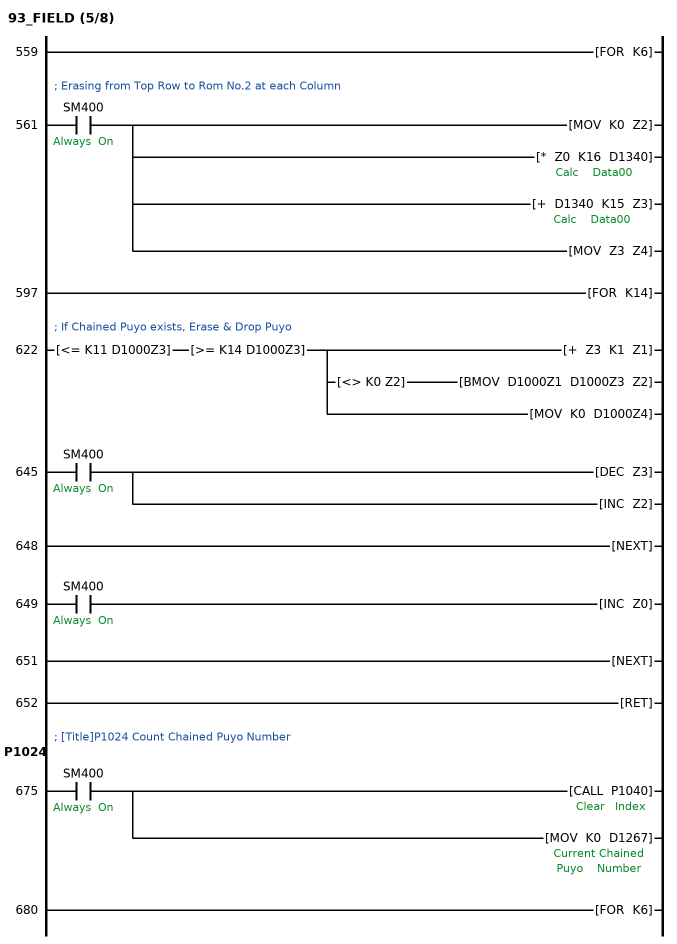
[picture p24: ladder of 93_FIELD, rungs at steps 559 to 680]
; Start Erasing at Column No.2 ,and End at No.7
559   FOR     K6
561   LD      SM400  ; Always  On
      MOV     K0 Z2
      *       Z0 K16 D1340
      +       D1340 K15 Z3
      MOV     Z3 Z4
; Erasing from Top Row to Rom No.2 at each Column
597   FOR     K14
; If Chained Puyo exists, Erase & Drop Puyo
622   LD<=    K11 D1000Z3
      AND>=   K14 D1000Z3
      +       Z3 K1 Z1
      MPS
      AND<>   K0 Z2
      BMOV    D1000Z1 D1000Z3 Z2
      MPP
      MOV     K0 D1000Z4
645   LD      SM400  ; Always  On
      DEC     Z3
      INC     Z2
648   NEXT
649   LD      SM400  ; Always  On
      INC     Z0
651   NEXT
652   RET
; [Title]P1024 Count Chained Puyo Number
      P1024
675   LD      SM400  ; Always  On
      CALL    P1040
      MOV     K0 D1267  ; Current Chained Puyo    Number
680   FOR     K6
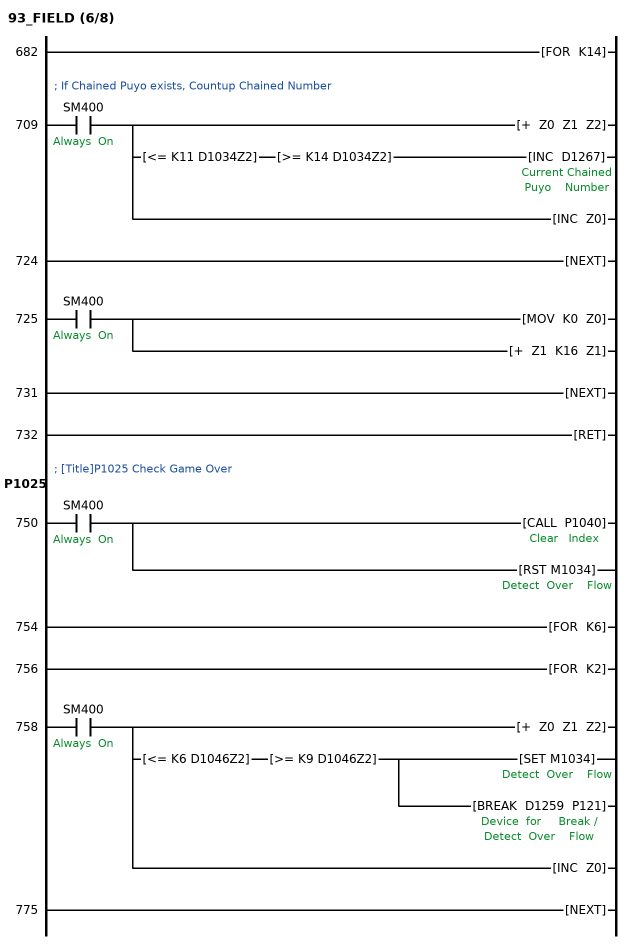
682   FOR     K14
; If Chained Puyo exists, Countup Chained Number
709   LD      SM400  ; Always  On
      +       Z0 Z1 Z2
      MPS
      AND<=   K11 D1034Z2
      AND>=   K14 D1034Z2
      INC     D1267
      MPP
      INC     Z0
724   NEXT
725   LD      SM400  ; Always  On
      MOV     K0 Z0
      +       Z1 K16 Z1
731   NEXT
732   RET
; [Title]P1025 Check Game Over
      P1025
750   LD      SM400  ; Always  On
      CALL    P1040
      RST     M1034  ; Detect  Over    Flow
754   FOR     K6
756   FOR     K2
758   LD      SM400  ; Always  On
      +       Z0 Z1 Z2
      MPS
      AND<=   K6 D1046Z2
      AND>=   K9 D1046Z2
      SET     M1034  ; Detect  Over    Flow
      BREAK   D1259 P121  ; Device  for     Break / Detect  Over    Flow
      MPP
      INC     Z0
775   NEXT
      P121
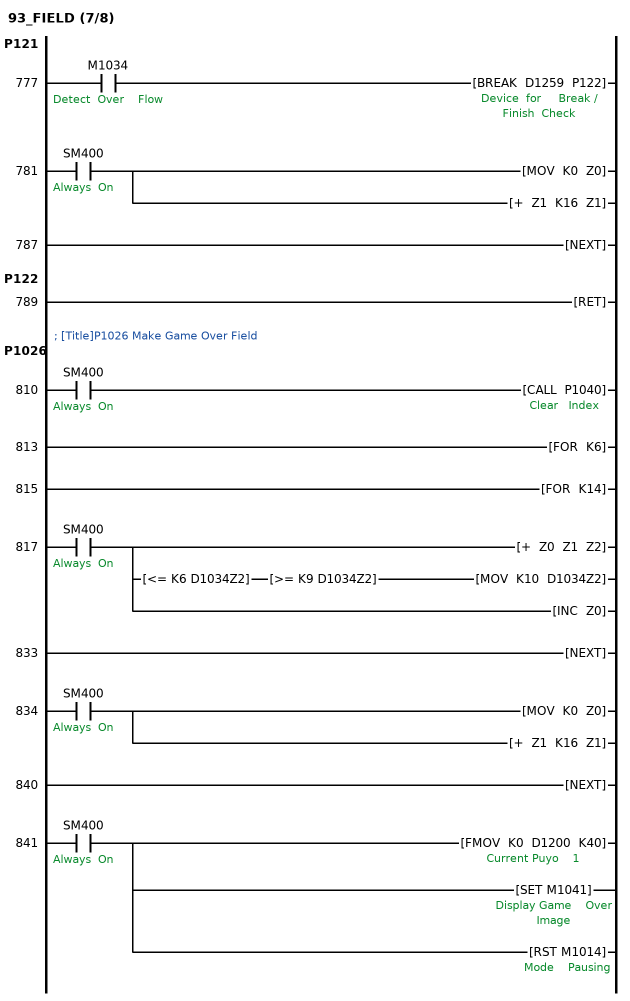
777   LD      M1034  ; Detect  Over    Flow
      BREAK   D1259 P122  ; Finish  Check
781   LD      SM400  ; Always  On
      MOV     K0 Z0
      +       Z1 K16 Z1
787   NEXT
      P122
789   RET
; [Title]P1026 Make Game Over Field
      P1026
810   LD      SM400  ; Always  On
      CALL    P1040
813   FOR     K6
815   FOR     K14
817   LD      SM400  ; Always  On
      +       Z0 Z1 Z2
      MPS
      AND<=   K6 D1034Z2
      AND>=   K9 D1034Z2
      MOV     K10 D1034Z2
      MPP
      INC     Z0
833   NEXT
834   LD      SM400  ; Always  On
      MOV     K0 Z0
      +       Z1 K16 Z1
840   NEXT
841   LD      SM400  ; Always  On
      FMOV    K0 D1200 K40  ; Current Puyo    1
      SET     M1041  ; Display Game    Over    Image
      RST     M1014  ; Mode    Pausing
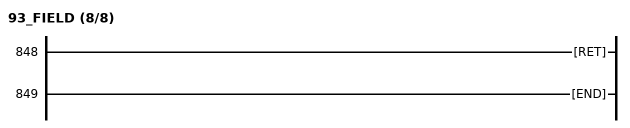
848   RET
849   END
END_PROGRAM

PROGRAM 94_MOVE  // Move Puyo Operation
; [Title]P1030 Move to Left Puyo
      P1030
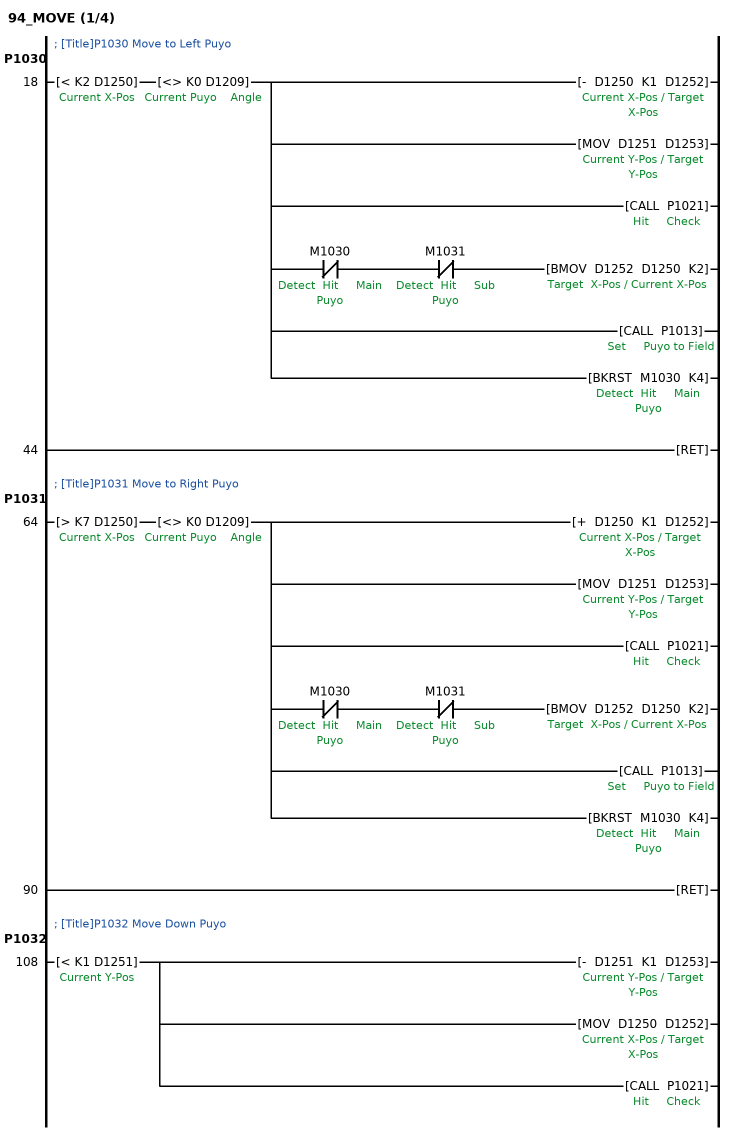
18    LD<     K2 D1250  ; Current X-Pos
      AND<>   K0 D1209  ; Current Puyo    Angle
      -       D1250 K1 D1252  ; Target  X-Pos
      MOV     D1251 D1253  ; Current Y-Pos / Target  Y-Pos
      CALL    P1021  ; Hit     Check
      MPS
      ANI     M1030  ; Detect  Hit     Main    Puyo
      ANI     M1031  ; Detect  Hit     Sub     Puyo
      BMOV    D1252 D1250 K2
      MPP
      CALL    P1013  ; Set     Puyo to Field
      BKRST   M1030 K4
44    RET
; [Title]P1031 Move to Right Puyo
      P1031
64    LD>     K7 D1250  ; Current X-Pos
      AND<>   K0 D1209  ; Current Puyo    Angle
      +       D1250 K1 D1252
      MOV     D1251 D1253
      CALL    P1021
      MPS
      ANI     M1030  ; Detect  Hit     Main    Puyo
      ANI     M1031  ; Detect  Hit     Sub     Puyo
      BMOV    D1252 D1250 K2
      MPP
      CALL    P1013
      BKRST   M1030 K4
90    RET
; [Title]P1032 Move Down Puyo
      P1032
108   LD<     K1 D1251  ; Current Y-Pos
      -       D1251 K1 D1253
      MOV     D1250 D1252
      CALL    P1021
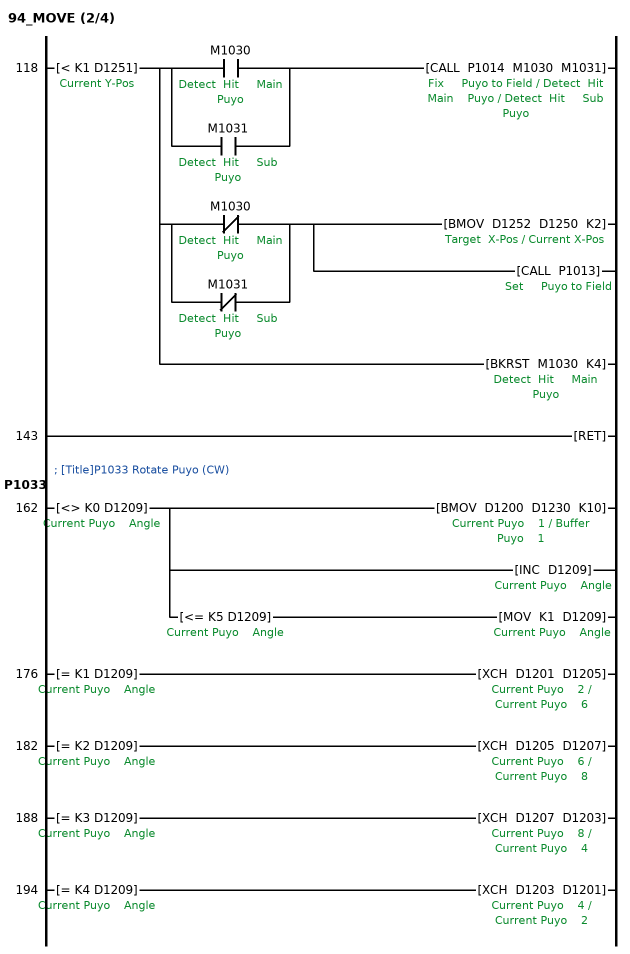
118   LD<     K1 D1251  ; Current Y-Pos
      MPS
      LD      M1030  ; Detect  Hit     Main    Puyo
      OR      M1031  ; Detect  Hit     Sub     Puyo
      ANB
      CALL    P1014 M1030 M1031  ; Fix     Puyo to Field
      MRD
      LDI     M1030  ; Detect  Hit     Main    Puyo
      ORI     M1031  ; Detect  Hit     Sub     Puyo
      ANB
      BMOV    D1252 D1250 K2
      CALL    P1013
      MPP
      BKRST   M1030 K4
143   RET
; [Title]P1033 Rotate Puyo (CW)
      P1033
162   LD<>    K0 D1209  ; Current Puyo    Angle
      BMOV    D1200 D1230 K10  ; Current Puyo    1 / Buffer  Puyo    1
      INC     D1209
      AND<=   K5 D1209  ; Current Puyo    Angle
      MOV     K1 D1209
176   LD=     K1 D1209  ; Current Puyo    Angle
      XCH     D1201 D1205  ; Current Puyo    2 / Current Puyo    6
182   LD=     K2 D1209  ; Current Puyo    Angle
      XCH     D1205 D1207  ; Current Puyo    8
188   LD=     K3 D1209  ; Current Puyo    Angle
      XCH     D1207 D1203  ; Current Puyo    4
194   LD=     K4 D1209  ; Current Puyo    Angle
      XCH     D1203 D1201
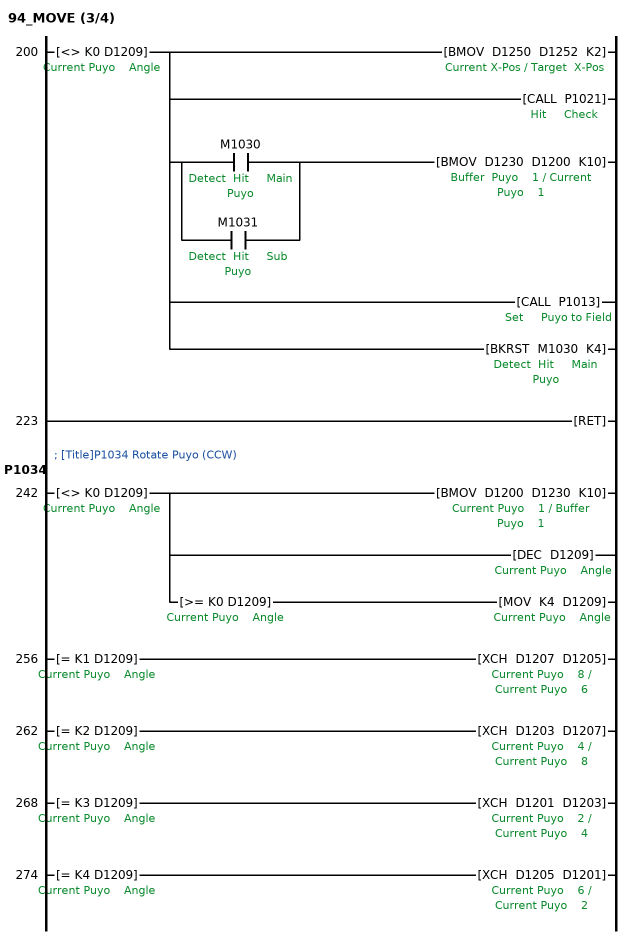
200   LD<>    K0 D1209  ; Current Puyo    Angle
      BMOV    D1250 D1252 K2
      CALL    P1021
      MPS
      LD      M1030  ; Detect  Hit     Main    Puyo
      OR      M1031  ; Detect  Hit     Sub     Puyo
      ANB
      BMOV    D1230 D1200 K10
      MPP
      CALL    P1013
      BKRST   M1030 K4
223   RET
; [Title]P1034 Rotate Puyo (CCW)
      P1034
242   LD<>    K0 D1209  ; Current Puyo    Angle
      BMOV    D1200 D1230 K10
      DEC     D1209
      AND>=   K0 D1209  ; Current Puyo    Angle
      MOV     K4 D1209
256   LD=     K1 D1209  ; Current Puyo    Angle
      XCH     D1207 D1205
262   LD=     K2 D1209  ; Current Puyo    Angle
      XCH     D1203 D1207
268   LD=     K3 D1209  ; Current Puyo    Angle
      XCH     D1201 D1203
274   LD=     K4 D1209  ; Current Puyo    Angle
      XCH     D1205 D1201
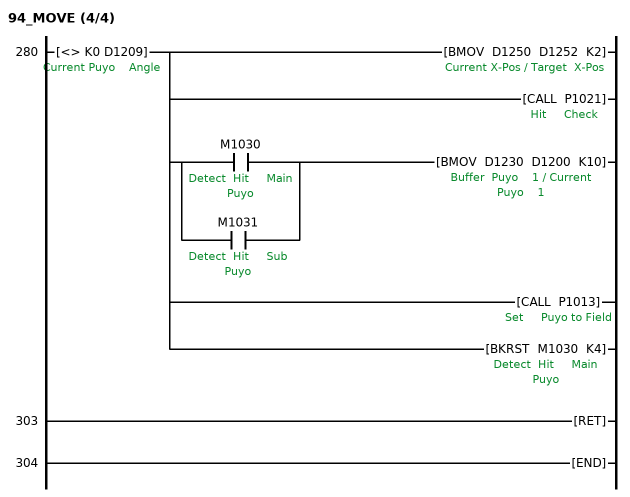
280   LD<>    K0 D1209  ; Current Puyo    Angle
      BMOV    D1250 D1252 K2
      CALL    P1021
      MPS
      LD      M1030  ; Detect  Hit     Main    Puyo
      OR      M1031  ; Detect  Hit     Sub     Puyo
      ANB
      BMOV    D1230 D1200 K10
      MPP
      CALL    P1013
      BKRST   M1030 K4
303   RET
304   END
END_PROGRAM

PROGRAM 02_GAME  // Game Main
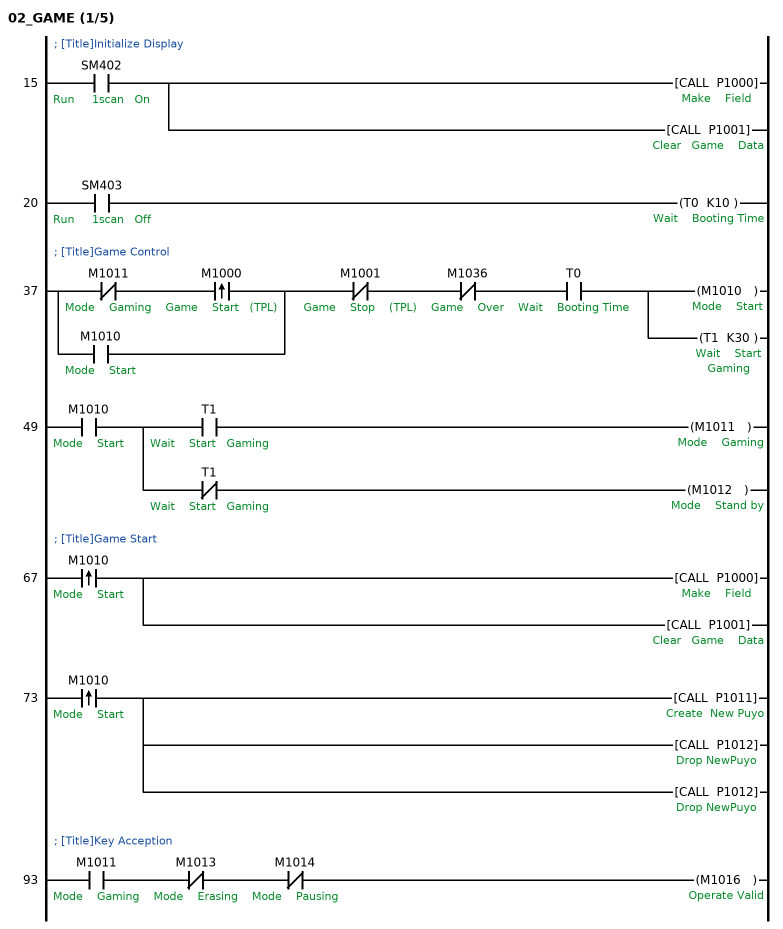
; [Title]Initialize Display
15    LD      SM402  ; Run     1scan   On
      CALL    P1000  ; Make    Field
      CALL    P1001  ; Clear   Game    Data
20    LD      SM403  ; Run     1scan   Off
      OUT     T0 K10  ; Wait    Booting Time
; [Title]Game Control
37    LDI     M1011  ; Mode    Gaming
      ANDP    M1000  ; Game    Start   (TPL)
      OR      M1010  ; Mode    Start
      ANI     M1001  ; Game    Stop    (TPL)
      ANI     M1036  ; Game    Over
      AND     T0  ; Wait    Booting Time
      OUT     M1010  ; Mode    Start
      OUT     T1 K30  ; Wait    Start   Gaming
49    LD      M1010  ; Mode    Start
      MPS
      AND     T1  ; Wait    Start   Gaming
      OUT     M1011  ; Mode    Gaming
      MPP
      ANI     T1  ; Wait    Start   Gaming
      OUT     M1012  ; Mode    Stand by
; [Title]Game Start
67    LDP     M1010  ; Mode    Start
      CALL    P1000
      CALL    P1001
73    LDP     M1010  ; Mode    Start
      CALL    P1011  ; Create  New Puyo
      CALL    P1012  ; Drop NewPuyo
      CALL    P1012
; [Title]Key Acception
93    LD      M1011  ; Mode    Gaming
      ANI     M1013  ; Mode    Erasing
      ANI     M1014  ; Mode    Pausing
      OUT     M1016  ; Operate Valid
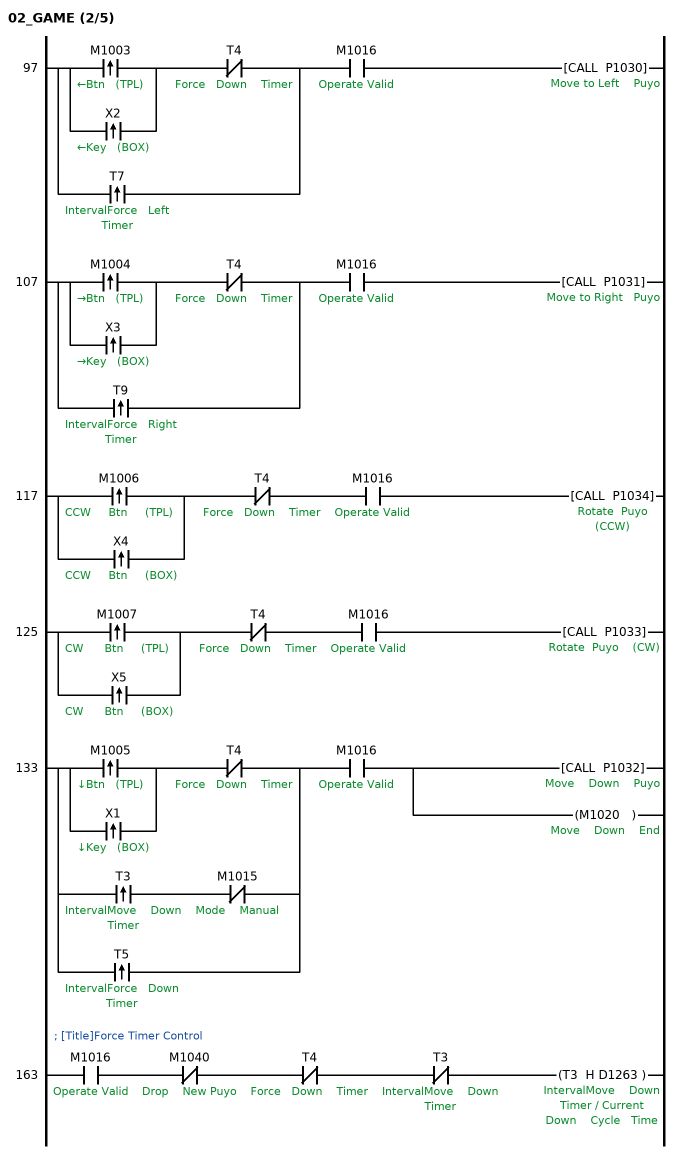
97    LDP     M1003  ; ←Btn   (TPL)
      ORP     X2  ; ←Key   (BOX)
      ANI     T4  ; Force   Down    Timer
      ORP     T7  ; IntervalForce   Left    Timer
      AND     M1016  ; Operate Valid
      CALL    P1030  ; Move to Left    Puyo
107   LDP     M1004  ; →Btn   (TPL)
      ORP     X3  ; →Key   (BOX)
      ANI     T4  ; Force   Down    Timer
      ORP     T9  ; IntervalForce   Right   Timer
      AND     M1016  ; Operate Valid
      CALL    P1031  ; Move to Right   Puyo
117   LDP     M1006  ; CCW     Btn     (TPL)
      ORP     X4  ; CCW     Btn     (BOX)
      ANI     T4  ; Force   Down    Timer
      AND     M1016  ; Operate Valid
      CALL    P1034  ; Rotate  Puyo    (CCW)
125   LDP     M1007  ; CW      Btn     (TPL)
      ORP     X5  ; CW      Btn     (BOX)
      ANI     T4  ; Force   Down    Timer
      AND     M1016  ; Operate Valid
      CALL    P1033  ; Rotate  Puyo    (CW)
133   LDP     M1005  ; ↓Btn   (TPL)
      ORP     X1  ; ↓Key   (BOX)
      ANI     T4  ; Force   Down    Timer
      LDP     T3  ; IntervalMove    Down    Timer
      ANI     M1015  ; Mode    Manual
      ORB
      ORP     T5  ; IntervalForce   Down    Timer
      AND     M1016  ; Operate Valid
      CALL    P1032  ; Move    Down    Puyo
      OUT     M1020  ; Move    Down    End
; [Title]Force Timer Control
163   LD      M1016  ; Operate Valid
      ANI     M1040  ; Drop    New Puyo
      ANI     T4  ; Force   Down    Timer
      ANI     T3  ; IntervalMove    Down    Timer
      OUTH    T3 D1263  ; IntervalMove    Down    Timer / Current Down    Cycle   Time
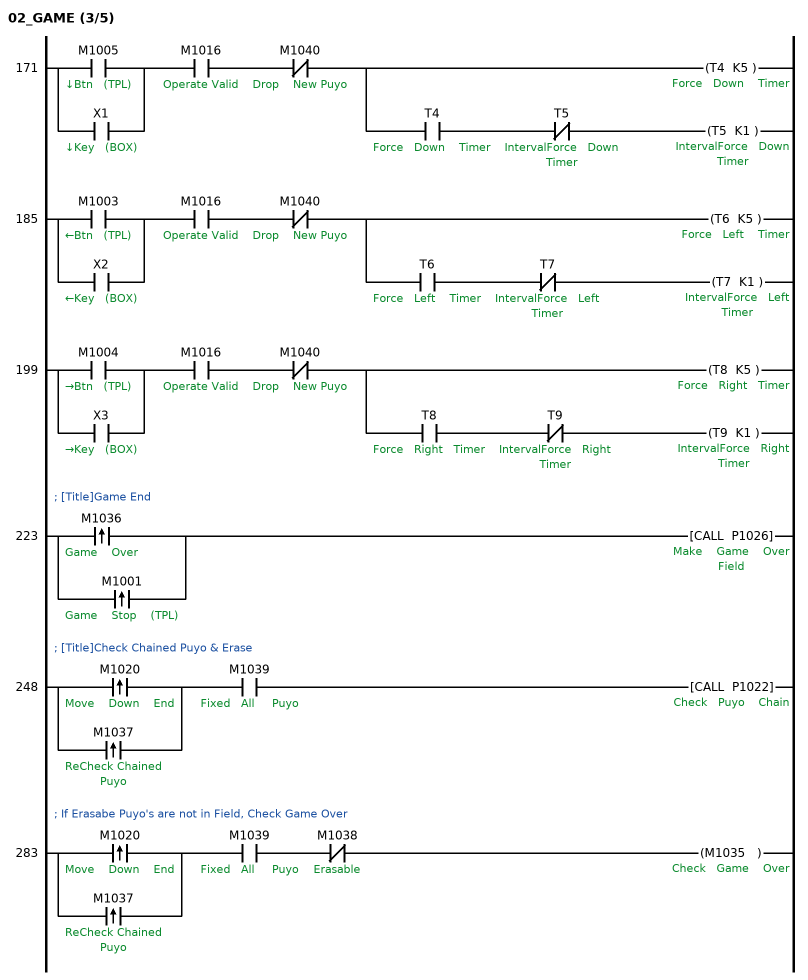
171   LD      M1005  ; ↓Btn   (TPL)
      OR      X1  ; ↓Key   (BOX)
      AND     M1016  ; Operate Valid
      ANI     M1040  ; Drop    New Puyo
      OUT     T4 K5  ; Force   Down    Timer
      AND     T4  ; Force   Down    Timer
      ANI     T5  ; IntervalForce   Down    Timer
      OUT     T5 K1  ; IntervalForce   Down    Timer
185   LD      M1003  ; ←Btn   (TPL)
      OR      X2  ; ←Key   (BOX)
      AND     M1016  ; Operate Valid
      ANI     M1040  ; Drop    New Puyo
      OUT     T6 K5  ; Force   Left    Timer
      AND     T6  ; Force   Left    Timer
      ANI     T7  ; IntervalForce   Left    Timer
      OUT     T7 K1  ; IntervalForce   Left    Timer
199   LD      M1004  ; →Btn   (TPL)
      OR      X3  ; →Key   (BOX)
      AND     M1016  ; Operate Valid
      ANI     M1040  ; Drop    New Puyo
      OUT     T8 K5  ; Force   Right   Timer
      AND     T8  ; Force   Right   Timer
      ANI     T9  ; IntervalForce   Right   Timer
      OUT     T9 K1  ; IntervalForce   Right   Timer
; [Title]Game End
223   LDP     M1036  ; Game    Over
      ORP     M1001  ; Game    Stop    (TPL)
      CALL    P1026  ; Make    Game    Over    Field
; [Title]Check Chained Puyo & Erase
248   LDP     M1020  ; Move    Down    End
      ORP     M1037  ; ReCheck Chained Puyo
      AND     M1039  ; Fixed   All     Puyo
      CALL    P1022  ; Check   Puyo    Chain
; If Erasabe Puyo's are not in Field, Check Game Over
283   LDP     M1020  ; Move    Down    End
      ORP     M1037  ; ReCheck Chained Puyo
      AND     M1039  ; Fixed   All     Puyo
      ANI     M1038  ; Erasable
      OUT     M1035  ; Check   Game    Over
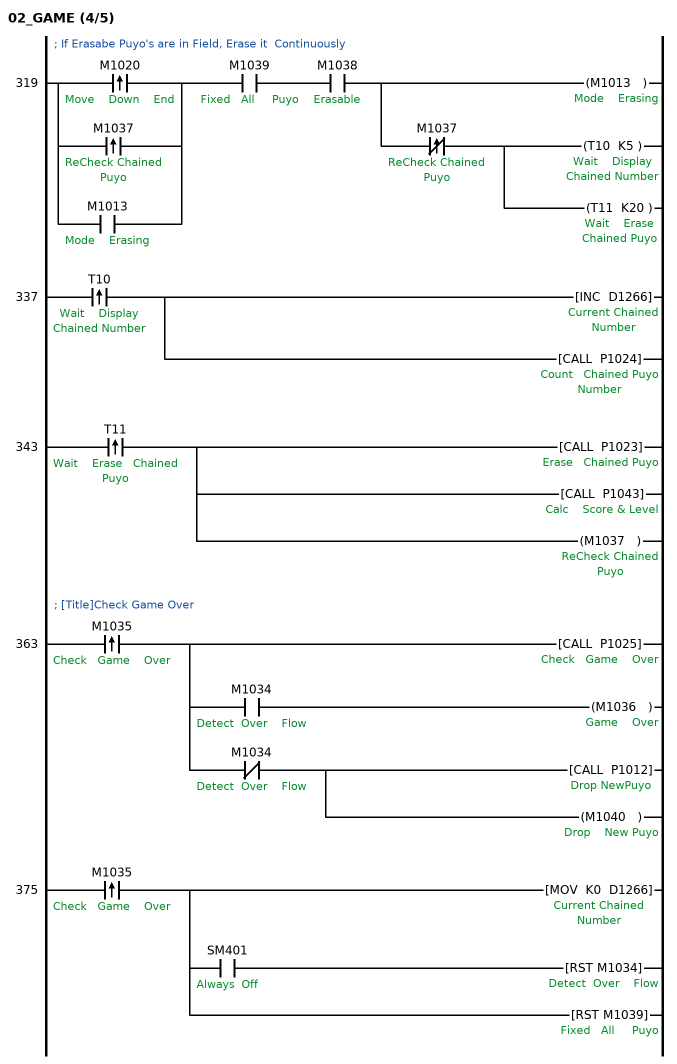
; If Erasabe Puyo's are in Field, Erase it  Continuously
319   LDP     M1020  ; Move    Down    End
      ORP     M1037  ; ReCheck Chained Puyo
      OR      M1013  ; Mode    Erasing
      AND     M1039  ; Fixed   All     Puyo
      AND     M1038  ; Erasable
      OUT     M1013  ; Mode    Erasing
      ANDPI   M1037  ; ReCheck Chained Puyo
      OUT     T10 K5  ; Wait    Display Chained Number
      OUT     T11 K20  ; Wait    Erase   Chained Puyo
337   LDP     T10  ; Wait    Display Chained Number
      INC     D1266  ; Current Chained Number
      CALL    P1024  ; Count   Chained Puyo    Number
343   LDP     T11  ; Wait    Erase   Chained Puyo
      CALL    P1023  ; Erase   Chained Puyo
      CALL    P1043  ; Calc    Score & Level
      OUT     M1037  ; ReCheck Chained Puyo
; [Title]Check Game Over
363   LDP     M1035  ; Check   Game    Over
      CALL    P1025  ; Check   Game    Over
      MPS
      AND     M1034  ; Detect  Over    Flow
      OUT     M1036  ; Game    Over
      MPP
      ANI     M1034  ; Detect  Over    Flow
      CALL    P1012
      OUT     M1040  ; Drop    New Puyo
375   LDP     M1035  ; Check   Game    Over
      MOV     K0 D1266
      MPS
      AND     SM401  ; Always  Off
      RST     M1034  ; Detect  Over    Flow
      MPP
      RST     M1039  ; Fixed   All     Puyo
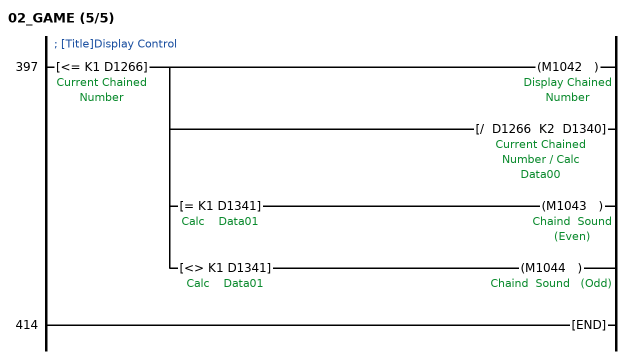
; [Title]Display Control
397   LD<=    K1 D1266  ; Current Chained Number
      OUT     M1042  ; Display Chained Number
      /       D1266 K2 D1340  ; Calc    Data00
      MPS
      AND=    K1 D1341  ; Calc    Data01
      OUT     M1043  ; Chaind  Sound   (Even)
      MPP
      AND<>   K1 D1341  ; Calc    Data01
      OUT     M1044  ; Chaind  Sound   (Odd)
414   END
END_PROGRAM

// device comments not shown above
D1034  ; Field   02, 02
M1017  ; Disable Free    Fall    Puyo
M1053  ; ==DBG== Trigger Setup   04
M1054  ; ==DBG== Trigger Setup   05
M1055  ; ==DBG== Trigger Setup   06
M1056  ; ==DBG== Trigger Setup   07
M1057  ; ==DBG== Trigger Setup   08
M1058  ; ==DBG== Trigger Setup   09
M1059  ; ==DBG== Trigger Setup   10
M1065  ; ==DBG== Trigger Puyo    06
M1066  ; ==DBG== Trigger Puyo    07
M1067  ; ==DBG== Trigger Puyo    08
M1068  ; ==DBG== Trigger Puyo    09
M1069  ; ==DBG== Trigger Puyo    10
M1077  ; ==DBG== Trigger Field   08
M1078  ; ==DBG== Trigger Field   09
M1079  ; ==DBG== Trigger Field   10
M1085  ; ==DBG== Trigger Move    06
M1086  ; ==DBG== Trigger Move    07
M1087  ; ==DBG== Trigger Move    08
M1088  ; ==DBG== Trigger Move    09
M1089  ; ==DBG== Trigger Move    10
M1095  ; ==DBG== Trigger Tools   06
M1096  ; ==DBG== Trigger Tools   07
M1097  ; ==DBG== Trigger Tools   08
M1098  ; ==DBG== Trigger Tools   09
M1099  ; ==DBG== Trigger Tools   10
P11  ; Create  New Puyo
D1001  ; Field   00, 01
D1002  ; Field   00, 02
D1003  ; Field   00, 03
D1004  ; Field   00, 04
D1005  ; Field   00, 05
D1006  ; Field   00, 06
D1007  ; Field   00, 07
D1008  ; Field   00, 08
D1009  ; Field   00, 09
D1010  ; Field   00, 10
D1011  ; Field   00, 11
D1012  ; Field   00, 12
D1013  ; Field   00, 13
D1014  ; Field   00, 14
D1015  ; Field   00, 15
D1016  ; Field   01, 00
D1017  ; Field   01, 01
D1018  ; Field   01, 02
D1019  ; Field   01, 03
D1020  ; Field   01, 04
D1021  ; Field   01, 05
D1022  ; Field   01, 06
D1023  ; Field   01, 07
D1024  ; Field   01, 08
D1025  ; Field   01, 09
D1026  ; Field   01, 10
D1027  ; Field   01, 11
D1028  ; Field   01, 12
D1029  ; Field   01, 13
D1030  ; Field   01, 14
D1031  ; Field   01, 15
D1033  ; Field   02, 01
D1035  ; Field   02, 03
D1036  ; Field   02, 04
D1037  ; Field   02, 05
D1038  ; Field   02, 06
D1039  ; Field   02, 07
D1040  ; Field   02, 08
D1041  ; Field   02, 09
D1042  ; Field   02, 10
D1043  ; Field   02, 11
D1044  ; Field   02, 12
D1045  ; Field   02, 13
D1046  ; Field   02, 14
D1047  ; Field   02, 15
D1048  ; Field   03, 00
D1049  ; Field   03, 01
D1050  ; Field   03, 02
D1051  ; Field   03, 03
D1052  ; Field   03, 04
D1053  ; Field   03, 05
D1054  ; Field   03, 06
D1055  ; Field   03, 07
D1056  ; Field   03, 08
D1057  ; Field   03, 09
D1058  ; Field   03, 10
D1059  ; Field   03, 11
D1060  ; Field   03, 12
D1061  ; Field   03, 13
D1062  ; Field   03, 14
D1063  ; Field   03, 15
D1064  ; Field   04, 00
D1065  ; Field   04, 01
D1066  ; Field   04, 02
D1067  ; Field   04, 03
D1068  ; Field   04, 04
D1069  ; Field   04, 05
D1070  ; Field   04, 06
D1071  ; Field   04, 07
D1072  ; Field   04, 08
D1073  ; Field   04, 09
D1074  ; Field   04, 10
D1075  ; Field   04, 11
D1076  ; Field   04, 12
D1077  ; Field   04, 13
D1078  ; Field   04, 14
D1079  ; Field   04, 15
D1080  ; Field   05, 00
D1081  ; Field   05, 01
D1082  ; Field   05, 02
D1083  ; Field   05, 03
D1084  ; Field   05, 04
D1085  ; Field   05, 05
D1086  ; Field   05, 06
D1087  ; Field   05, 07
D1088  ; Field   05, 08
D1089  ; Field   05, 09
D1090  ; Field   05, 10
D1091  ; Field   05, 11
D1092  ; Field   05, 12
D1093  ; Field   05, 13
D1094  ; Field   05, 14
D1095  ; Field   05, 15
D1096  ; Field   06, 00
D1097  ; Field   06, 01
D1098  ; Field   06, 02
D1099  ; Field   06, 03
D1100  ; Field   06, 04
D1101  ; Field   06, 05
D1102  ; Field   06, 06
D1103  ; Field   06, 07
D1104  ; Field   06, 08
D1105  ; Field   06, 09
D1106  ; Field   06, 10
D1107  ; Field   06, 11
D1108  ; Field   06, 12
D1109  ; Field   06, 13
D1110  ; Field   06, 14
D1111  ; Field   06, 15
D1112  ; Field   07, 00
D1113  ; Field   07, 01
D1114  ; Field   07, 02
D1115  ; Field   07, 03
D1116  ; Field   07, 04
D1117  ; Field   07, 05
D1118  ; Field   07, 06
D1119  ; Field   07, 07
D1120  ; Field   07, 08
D1121  ; Field   07, 09
D1122  ; Field   07, 10
D1123  ; Field   07, 11
D1124  ; Field   07, 12
D1125  ; Field   07, 13
D1126  ; Field   07, 14
D1127  ; Field   07, 15
D1129  ; Field   08, 01
D1130  ; Field   08, 02
D1131  ; Field   08, 03
D1132  ; Field   08, 04
D1133  ; Field   08, 05
D1134  ; Field   08, 06
D1135  ; Field   08, 07
D1136  ; Field   08, 08
D1137  ; Field   08, 09
D1138  ; Field   08, 10
D1139  ; Field   08, 11
D1140  ; Field   08, 12
D1141  ; Field   08, 13
D1142  ; Field   08, 14
D1143  ; Field   08, 15
D1144  ; Field   09, 00
D1145  ; Field   09, 01
D1146  ; Field   09, 02
D1147  ; Field   09, 03
D1148  ; Field   09, 04
D1149  ; Field   09, 05
D1150  ; Field   09, 06
D1151  ; Field   09, 07
D1152  ; Field   09, 08
D1153  ; Field   09, 09
D1154  ; Field   09, 10
D1155  ; Field   09, 11
D1156  ; Field   09, 12
D1157  ; Field   09, 13
D1158  ; Field   09, 14
D1159  ; Field   09, 15
D1202  ; Current Puyo    3
D1206  ; Current Puyo    7
D1208  ; Current Puyo    9
D1211  ; Reserve Puyo    1-2
D1212  ; Reserve Puyo    1-3
D1213  ; Reserve Puyo    1-4
D1214  ; Reserve Puyo    1-5
D1215  ; Reserve Puyo    1-6
D1216  ; Reserve Puyo    1-7
D1217  ; Reserve Puyo    1-8
D1218  ; Reserve Puyo    1-9
D1219  ; Reserve Puyo    Angle 1
D1221  ; Reserve Puyo    2-2
D1222  ; Reserve Puyo    2-3
D1223  ; Reserve Puyo    2-4
D1224  ; Reserve Puyo    2-5
D1225  ; Reserve Puyo    2-6
D1226  ; Reserve Puyo    2-7
D1227  ; Reserve Puyo    2-8
D1228  ; Reserve Puyo    2-9
D1231  ; Buffer  Puyo    2
D1232  ; Buffer  Puyo    3
D1233  ; Buffer  Puyo    4
D1234  ; Buffer  Puyo    5
D1235  ; Buffer  Puyo    6
D1236  ; Buffer  Puyo    7
D1237  ; Buffer  Puyo    8
D1238  ; Buffer  Puyo    9
D1239  ; Buffer  Puyo    Angle
D1261  ; Current Score   (H)
D1280  ; 9's     Field   Address Offset01
D1281  ; 9's     Field   Address Offset02
D1282  ; 9's     Field   Address Offset03
D1283  ; 9's     Field   Address Offset04
D1284  ; 9's     Field   Address Offset05
D1285  ; 9's     Field   Address Offset06
D1286  ; 9's     Field   Address Offset07
D1287  ; 9's     Field   Address Offset08
D1288  ; 9's     Field   Address Offset09
D1302  ; Next    Puyo    Order   03
D1303  ; Next    Puyo    Order   04
D1304  ; Next    Puyo    Order   05
D1305  ; Next    Puyo    Order   06
D1306  ; Next    Puyo    Order   07
D1307  ; Next    Puyo    Order   08
D1308  ; Next    Puyo    Order   09
D1309  ; Next    Puyo    Order   10
D1310  ; Next    Puyo    Order   11
D1311  ; Next    Puyo    Order   12
D1312  ; Next    Puyo    Order   13
D1313  ; Next    Puyo    Order   14
D1314  ; Next    Puyo    Order   15
D1321  ; Puyo    Order   Array   02
D1322  ; Puyo    Order   Array   03
D1323  ; Puyo    Order   Array   04
D1324  ; Puyo    Order   Array   05
D1325  ; Puyo    Order   Array   06
D1326  ; Puyo    Order   Array   07
D1327  ; Puyo    Order   Array   08
D1328  ; Puyo    Order   Array   09
D1329  ; Puyo    Order   Array   10
D1330  ; Puyo    Order   Array   11
D1331  ; Puyo    Order   Array   12
D1332  ; Puyo    Order   Array   13
D1333  ; Puyo    Order   Array   14
D1334  ; Puyo    Order   Array   15
D1335  ; Puyo    Order   Array   16
D1346  ; Calc    Data06
D1347  ; Calc    Data07
D1348  ; Calc    Data08
D1349  ; Calc    Data09
D3001  ; Puyo    Data    GG 2
D3002  ; Puyo    Data    GG 3
D3003  ; Puyo    Data    GG 4
D3006  ; Puyo    Data    GG 7
D3007  ; Puyo    Data    GG 8
D3008  ; Puyo    Data    GG 9
D3009  ; Puyo    Data    GR 1
D3010  ; Puyo    Data    GR 2
D3011  ; Puyo    Data    GR 3
D3012  ; Puyo    Data    GR 4
D3015  ; Puyo    Data    GR 7
D3016  ; Puyo    Data    GR 8
D3017  ; Puyo    Data    GR 9
D3018  ; Puyo    Data    GB 1
D3019  ; Puyo    Data    GB 2
D3020  ; Puyo    Data    GB 3
D3021  ; Puyo    Data    GB 4
D3024  ; Puyo    Data    GB 7
D3025  ; Puyo    Data    GB 8
D3026  ; Puyo    Data    GB 9
D3027  ; Puyo    Data    GY 1
D3028  ; Puyo    Data    GY 2
D3029  ; Puyo    Data    GY 3
D3030  ; Puyo    Data    GY 4
D3033  ; Puyo    Data    GY 7
D3034  ; Puyo    Data    GY 8
D3035  ; Puyo    Data    GY 9
D3036  ; Puyo    Data    RG 1
D3037  ; Puyo    Data    RG 2
D3038  ; Puyo    Data    RG 3
D3039  ; Puyo    Data    RG 4
D3042  ; Puyo    Data    RG 7
D3043  ; Puyo    Data    RG 8
D3044  ; Puyo    Data    RG 9
D3045  ; Puyo    Data    RR 1
D3046  ; Puyo    Data    RR 2
D3047  ; Puyo    Data    RR 3
D3048  ; Puyo    Data    RR 4
D3051  ; Puyo    Data    RR 7
D3052  ; Puyo    Data    RR 8
D3053  ; Puyo    Data    RR 9
D3054  ; Puyo    Data    RB 1
D3055  ; Puyo    Data    RB 2
D3056  ; Puyo    Data    RB 3
D3057  ; Puyo    Data    RB 4
D3060  ; Puyo    Data    RB 7
D3061  ; Puyo    Data    RB 8
D3062  ; Puyo    Data    RB 9
D3063  ; Puyo    Data    RY 1
D3064  ; Puyo    Data    RY 2
D3065  ; Puyo    Data    RY 3
D3066  ; Puyo    Data    RY 4
D3069  ; Puyo    Data    RY 7
D3070  ; Puyo    Data    RY 8
D3071  ; Puyo    Data    RY 9
D3072  ; Puyo    Data    BG 1
D3073  ; Puyo    Data    BG 2
D3074  ; Puyo    Data    BG 3
D3075  ; Puyo    Data    BG 4
D3078  ; Puyo    Data    BG 7
D3079  ; Puyo    Data    BG 8
D3080  ; Puyo    Data    BG 9
D3081  ; Puyo    Data    BR 1
D3082  ; Puyo    Data    BR 2
D3083  ; Puyo    Data    BR 3
D3084  ; Puyo    Data    BR 4
D3087  ; Puyo    Data    BR 7
D3088  ; Puyo    Data    BR 8
D3089  ; Puyo    Data    BR 9
D3090  ; Puyo    Data    BB 1
D3091  ; Puyo    Data    BB 2
D3092  ; Puyo    Data    BB 3
D3093  ; Puyo    Data    BB 4
D3096  ; Puyo    Data    BB 7
D3097  ; Puyo    Data    BB 8
D3098  ; Puyo    Data    BB 9
D3099  ; Puyo    Data    BY 1
D3100  ; Puyo    Data    BY 2
D3101  ; Puyo    Data    BY 3
D3102  ; Puyo    Data    BY 4
D3105  ; Puyo    Data    BY 7
D3106  ; Puyo    Data    BY 8
D3107  ; Puyo    Data    BY 9
D3108  ; Puyo    Data    YG 1
D3109  ; Puyo    Data    YG 2
D3110  ; Puyo    Data    YG 3
D3111  ; Puyo    Data    YG 4
D3114  ; Puyo    Data    YG 7
D3115  ; Puyo    Data    YG 8
D3116  ; Puyo    Data    YG 9
D3117  ; Puyo    Data    YR 1
D3118  ; Puyo    Data    YR 2
D3119  ; Puyo    Data    YR 3
D3120  ; Puyo    Data    YR 4
D3123  ; Puyo    Data    YR 7
D3124  ; Puyo    Data    YR 8
D3125  ; Puyo    Data    YR 9
D3126  ; Puyo    Data    YB 1
D3127  ; Puyo    Data    YB 2
D3128  ; Puyo    Data    YB 3
D3129  ; Puyo    Data    YB 4
D3132  ; Puyo    Data    YB 7
D3133  ; Puyo    Data    YB 8
D3134  ; Puyo    Data    YB 9
D3135  ; Puyo    Data    YY 1
D3136  ; Puyo    Data    YY 2
D3137  ; Puyo    Data    YY 3
D3138  ; Puyo    Data    YY 4
D3141  ; Puyo    Data    YY 7
D3142  ; Puyo    Data    YY 8
D3143  ; Puyo    Data    YY 9
D5001  ; 1to16   Asc     Order   Num02
D5002  ; 1to16   Asc     Order   Num03
D5003  ; 1to16   Asc     Order   Num04
D5004  ; 1to16   Asc     Order   Num05
D5005  ; 1to16   Asc     Order   Num06
D5006  ; 1to16   Asc     Order   Num07
D5007  ; 1to16   Asc     Order   Num08
D5008  ; 1to16   Asc     Order   Num09
D5009  ; 1to16   Asc     Order   Num10
D5010  ; 1to16   Asc     Order   Num11
D5011  ; 1to16   Asc     Order   Num12
D5012  ; 1to16   Asc     Order   Num13
D5013  ; 1to16   Asc     Order   Num14
D5014  ; 1to16   Asc     Order   Num15
D5015  ; 1to16   Asc     Order   Num16
D6200  ; Bottom  Puyo    Address
